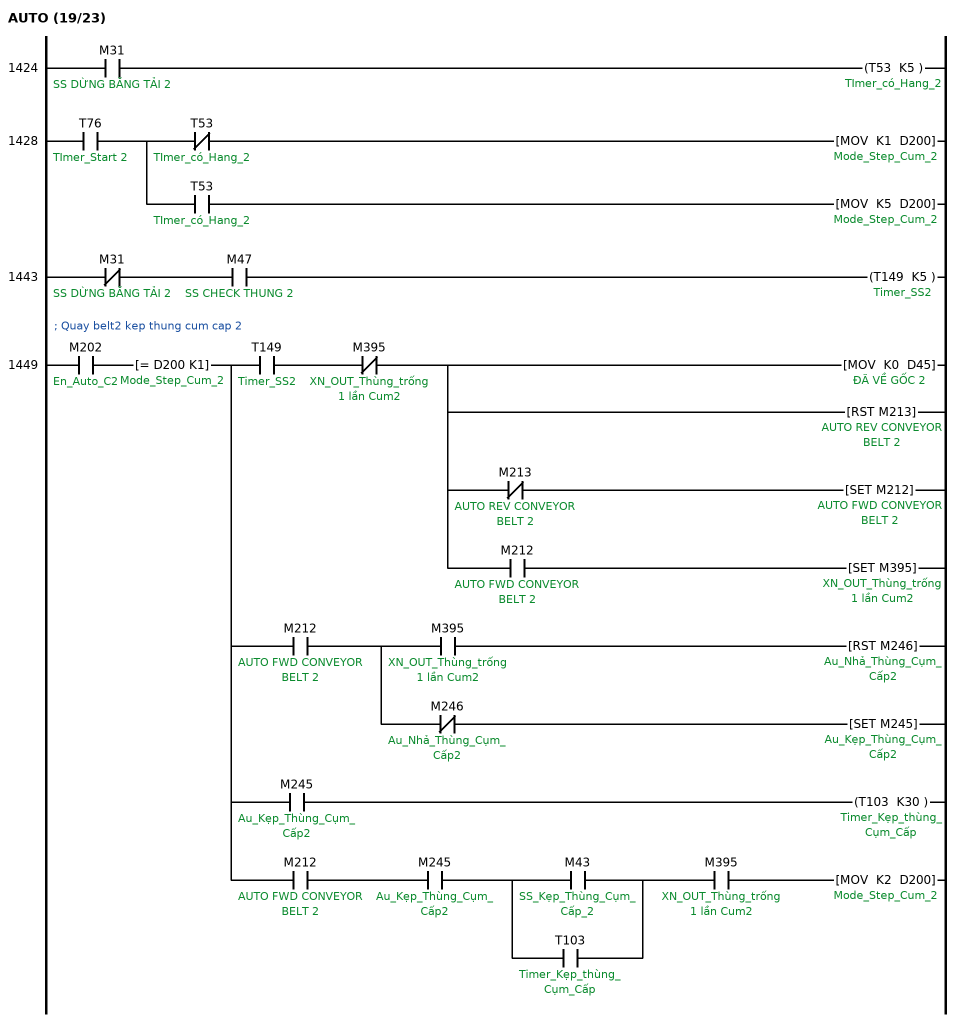
1424  LD      M31  ; SS DỪNG BĂNG TẢI 2
      OUT     T53 K5  ; TImer_có_Hang_2
1428  LD      T76  ; TImer_Start 2
      MPS
      ANI     T53  ; TImer_có_Hang_2
      MOV     K1 D200
      MPP
      AND     T53  ; TImer_có_Hang_2
      MOV     K5 D200
1443  LDI     M31  ; SS DỪNG BĂNG TẢI 2
      AND     M47  ; SS CHECK THUNG 2
      OUT     T149 K5  ; Timer_SS2
; Quay belt2 kep thung cum cap 2
1449  LD      M202  ; En_Auto_C2
      AND=    D200 K1  ; Mode_Step_Cum_2
      MPS
      AND     T149  ; Timer_SS2
      ANI     M395  ; XN_OUT_Thùng_trống 1 lần Cum2
      MOV     K0 D45
      RST     M213  ; AUTO REV CONVEYOR BELT 2
      MPS
      ANI     M213  ; AUTO REV CONVEYOR BELT 2
      SET     M212  ; AUTO FWD CONVEYOR BELT 2
      MPP
      AND     M212  ; AUTO FWD CONVEYOR BELT 2
      SET     M395  ; XN_OUT_Thùng_trống 1 lần Cum2
      MRD
      AND     M212  ; AUTO FWD CONVEYOR BELT 2
      MPS
      AND     M395  ; XN_OUT_Thùng_trống 1 lần Cum2
      RST     M246  ; Au_Nhả_Thùng_Cụm_Cấp2
      MPP
      ANI     M246  ; Au_Nhả_Thùng_Cụm_Cấp2
      SET     M245  ; Au_Kẹp_Thùng_Cụm_Cấp2
      MRD
      AND     M245  ; Au_Kẹp_Thùng_Cụm_Cấp2
      OUT     T103 K30  ; Timer_Kẹp_thùng_Cụm_Cấp
      MPP
      AND     M212  ; AUTO FWD CONVEYOR BELT 2
      AND     M245  ; Au_Kẹp_Thùng_Cụm_Cấp2
      LD      M43  ; SS_Kẹp_Thùng_Cụm_Cấp_2
      OR      T103  ; Timer_Kẹp_thùng_Cụm_Cấp
      ANB
      AND     M395  ; XN_OUT_Thùng_trống 1 lần Cum2
      MOV     K2 D200
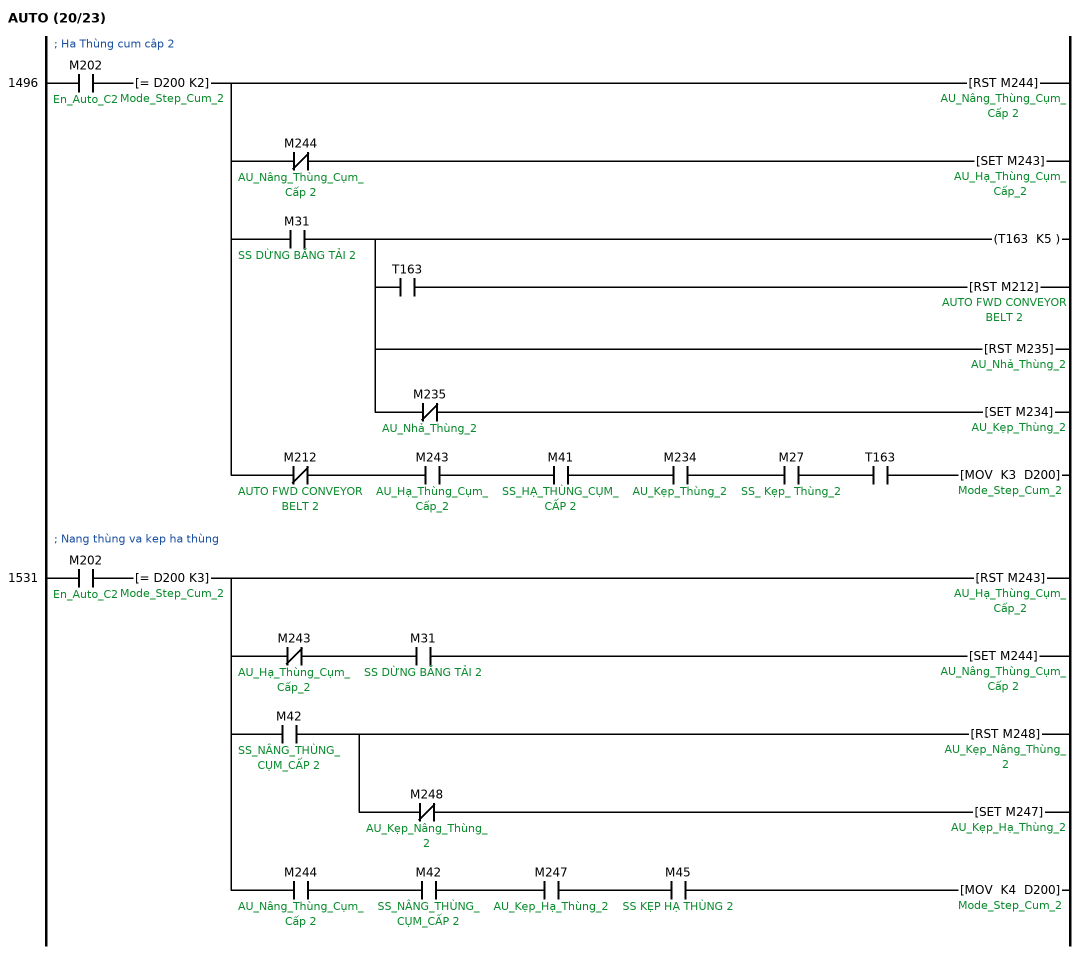
; Ha Thùng cum câp 2
1496  LD      M202  ; En_Auto_C2
      AND=    D200 K2  ; Mode_Step_Cum_2
      RST     M244  ; AU_Nâng_Thùng_Cụm_Cấp 2
      MPS
      ANI     M244  ; AU_Nâng_Thùng_Cụm_Cấp 2
      SET     M243  ; AU_Hạ_Thùng_Cụm_Cấp_2
      MRD
      AND     M31  ; SS DỪNG BĂNG TẢI 2
      OUT     T163 K5
      MPS
      AND     T163
      RST     M212  ; AUTO FWD CONVEYOR BELT 2
      MPP
      RST     M235  ; AU_Nhả_Thùng_2
      ANI     M235  ; AU_Nhả_Thùng_2
      SET     M234  ; AU_Kẹp_Thùng_2
      MPP
      ANI     M212  ; AUTO FWD CONVEYOR BELT 2
      AND     M243  ; AU_Hạ_Thùng_Cụm_Cấp_2
      AND     M41  ; SS_HẠ_THÙNG_CỤM_CẤP 2
      AND     M234  ; AU_Kẹp_Thùng_2
      AND     M27  ; SS_ Kẹp_ Thùng_2
      AND     T163
      MOV     K3 D200
; Nang thùng va kep ha thùng
1531  LD      M202  ; En_Auto_C2
      AND=    D200 K3  ; Mode_Step_Cum_2
      RST     M243  ; AU_Hạ_Thùng_Cụm_Cấp_2
      MPS
      ANI     M243  ; AU_Hạ_Thùng_Cụm_Cấp_2
      AND     M31  ; SS DỪNG BĂNG TẢI 2
      SET     M244  ; AU_Nâng_Thùng_Cụm_Cấp 2
      MRD
      AND     M42  ; SS_NÂNG_THÙNG_CỤM_CẤP 2
      RST     M248  ; AU_Kẹp_Nâng_Thùng_2
      ANI     M248  ; AU_Kẹp_Nâng_Thùng_2
      SET     M247  ; AU_Kẹp_Hạ_Thùng_2
      MPP
      AND     M244  ; AU_Nâng_Thùng_Cụm_Cấp 2
      AND     M42  ; SS_NÂNG_THÙNG_CỤM_CẤP 2
      AND     M247  ; AU_Kẹp_Hạ_Thùng_2
      AND     M45  ; SS KẸP HẠ THÙNG 2
      MOV     K4 D200
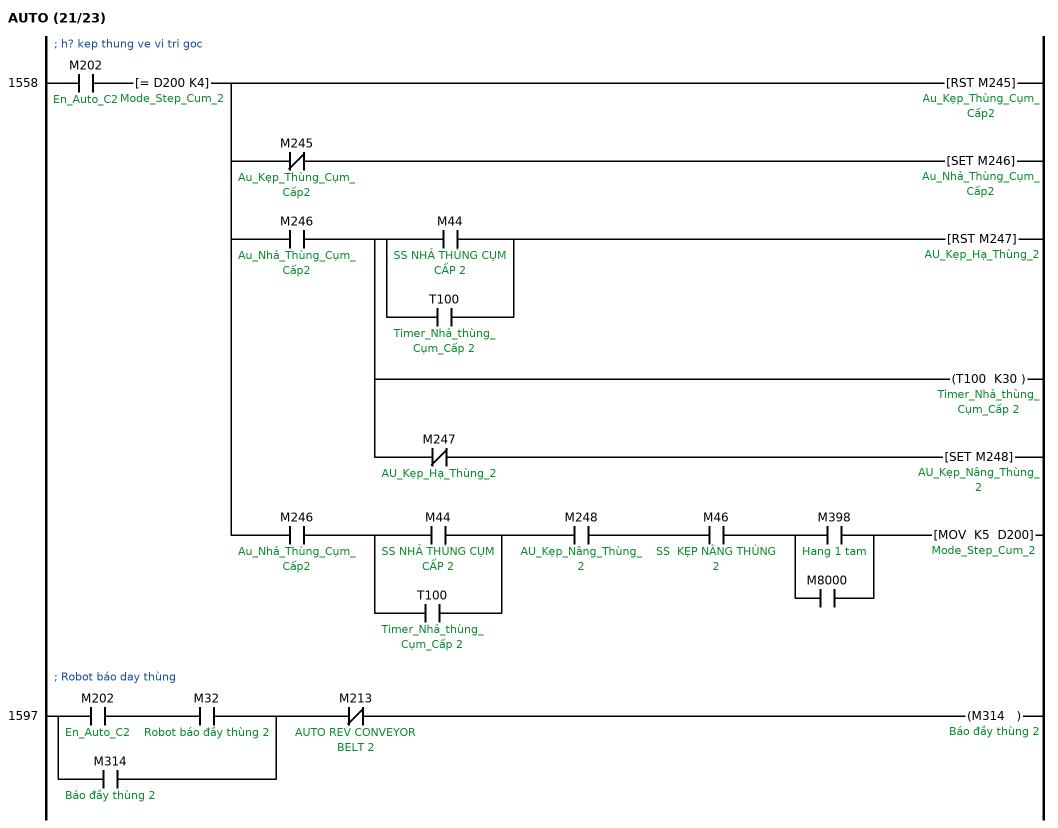
; h? kep thung ve vi tri goc
1558  LD      M202  ; En_Auto_C2
      AND=    D200 K4  ; Mode_Step_Cum_2
      RST     M245  ; Au_Kẹp_Thùng_Cụm_Cấp2
      MPS
      ANI     M245  ; Au_Kẹp_Thùng_Cụm_Cấp2
      SET     M246  ; Au_Nhả_Thùng_Cụm_Cấp2
      MRD
      AND     M246  ; Au_Nhả_Thùng_Cụm_Cấp2
      MPS
      LD      M44  ; SS NHẢ THÙNG CỤM CẤP 2
      OR      T100  ; Timer_Nhả_thùng_Cụm_Cấp 2
      ANB
      RST     M247  ; AU_Kẹp_Hạ_Thùng_2
      MPP
      OUT     T100 K30  ; Timer_Nhả_thùng_Cụm_Cấp 2
      ANI     M247  ; AU_Kẹp_Hạ_Thùng_2
      SET     M248  ; AU_Kẹp_Nâng_Thùng_2
      MPP
      AND     M246  ; Au_Nhả_Thùng_Cụm_Cấp2
      LD      M44  ; SS NHẢ THÙNG CỤM CẤP 2
      OR      T100  ; Timer_Nhả_thùng_Cụm_Cấp 2
      ANB
      AND     M248  ; AU_Kẹp_Nâng_Thùng_2
      AND     M46  ; SS  KẸP NÂNG THÙNG 2
      LD      M398  ; Hang 1 tam
      OR      M8000
      ANB
      MOV     K5 D200
; Robot báo day thùng
1597  LD      M202  ; En_Auto_C2
      AND     M32  ; Robot báo đầy thùng 2
      OR      M314  ; Báo đầy thùng 2
      ANI     M213  ; AUTO REV CONVEYOR BELT 2
      OUT     M314  ; Báo đầy thùng 2
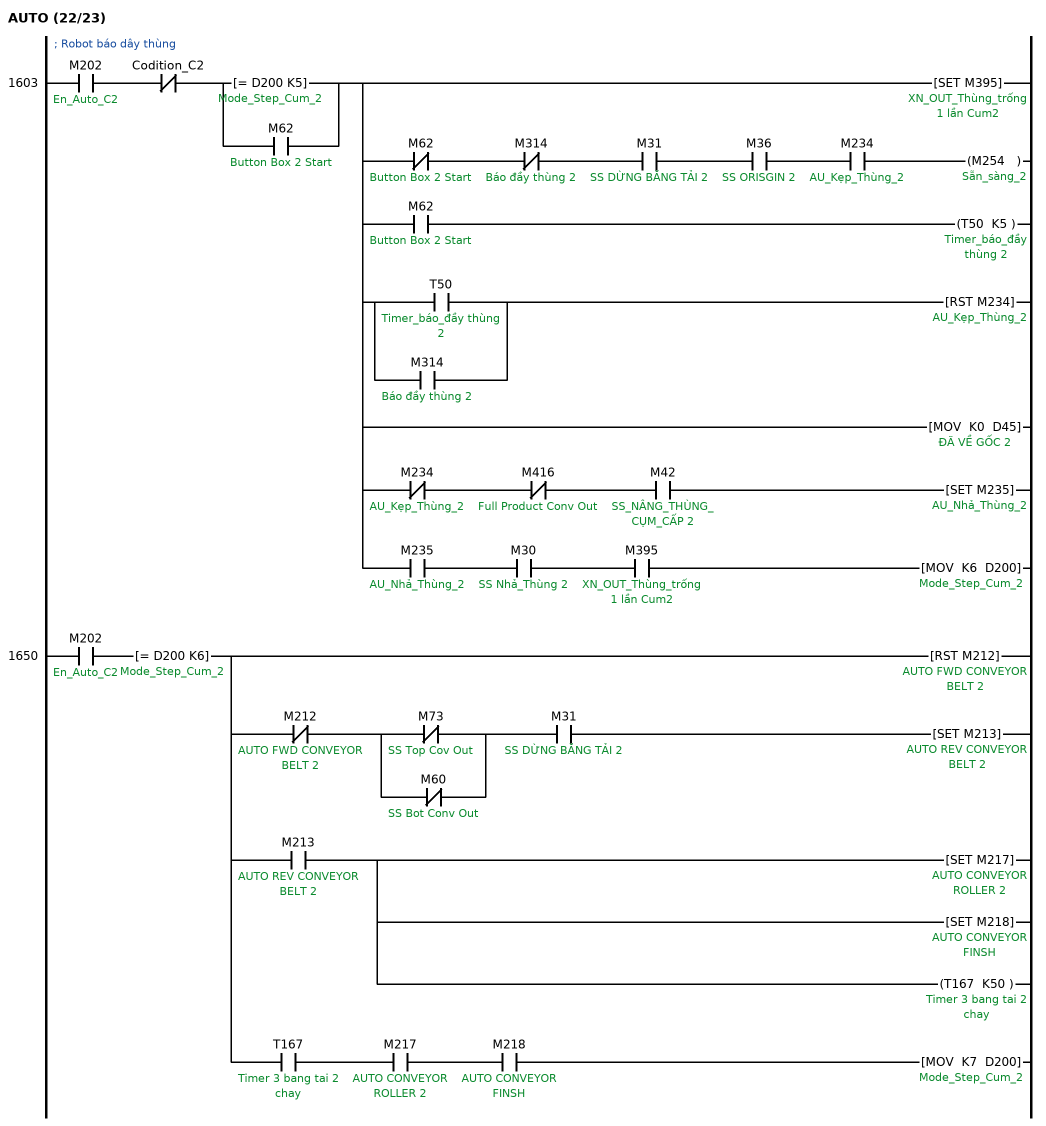
; Robot báo dây thùng
1603  LD      M202  ; En_Auto_C2
      ANI     Codition_C2
      LD=     D200 K5  ; Mode_Step_Cum_2
      OR      M62  ; Button Box 2 Start
      ANB
      SET     M395  ; XN_OUT_Thùng_trống 1 lần Cum2
      MPS
      ANI     M62  ; Button Box 2 Start
      ANI     M314  ; Báo đầy thùng 2
      AND     M31  ; SS DỪNG BĂNG TẢI 2
      AND     M36  ; SS ORISGIN 2
      AND     M234  ; AU_Kẹp_Thùng_2
      OUT     M254  ; Sẵn_sàng_2
      MRD
      AND     M62  ; Button Box 2 Start
      OUT     T50 K5  ; Timer_báo_đầy thùng 2
      MRD
      LD      T50  ; Timer_báo_đầy thùng 2
      OR      M314  ; Báo đầy thùng 2
      ANB
      RST     M234  ; AU_Kẹp_Thùng_2
      MPP
      MOV     K0 D45
      MPS
      ANI     M234  ; AU_Kẹp_Thùng_2
      ANI     M416  ; Full Product Conv Out
      AND     M42  ; SS_NÂNG_THÙNG_CỤM_CẤP 2
      SET     M235  ; AU_Nhả_Thùng_2
      MPP
      AND     M235  ; AU_Nhả_Thùng_2
      AND     M30  ; SS Nhả_Thùng 2
      AND     M395  ; XN_OUT_Thùng_trống 1 lần Cum2
      MOV     K6 D200
1650  LD      M202  ; En_Auto_C2
      AND=    D200 K6  ; Mode_Step_Cum_2
      RST     M212  ; AUTO FWD CONVEYOR BELT 2
      MPS
      ANI     M212  ; AUTO FWD CONVEYOR BELT 2
      LDI     M73  ; SS Top Cov Out
      ORI     M60  ; SS Bot Conv Out
      ANB
      AND     M31  ; SS DỪNG BĂNG TẢI 2
      SET     M213  ; AUTO REV CONVEYOR BELT 2
      MRD
      AND     M213  ; AUTO REV CONVEYOR BELT 2
      SET     M217  ; AUTO CONVEYOR ROLLER 2
      SET     M218  ; AUTO CONVEYOR FINSH
      OUT     T167 K50  ; Timer 3 bang tai 2 chay
      MPP
      AND     T167  ; Timer 3 bang tai 2 chay
      AND     M217  ; AUTO CONVEYOR ROLLER 2
      AND     M218  ; AUTO CONVEYOR FINSH
      MOV     K7 D200
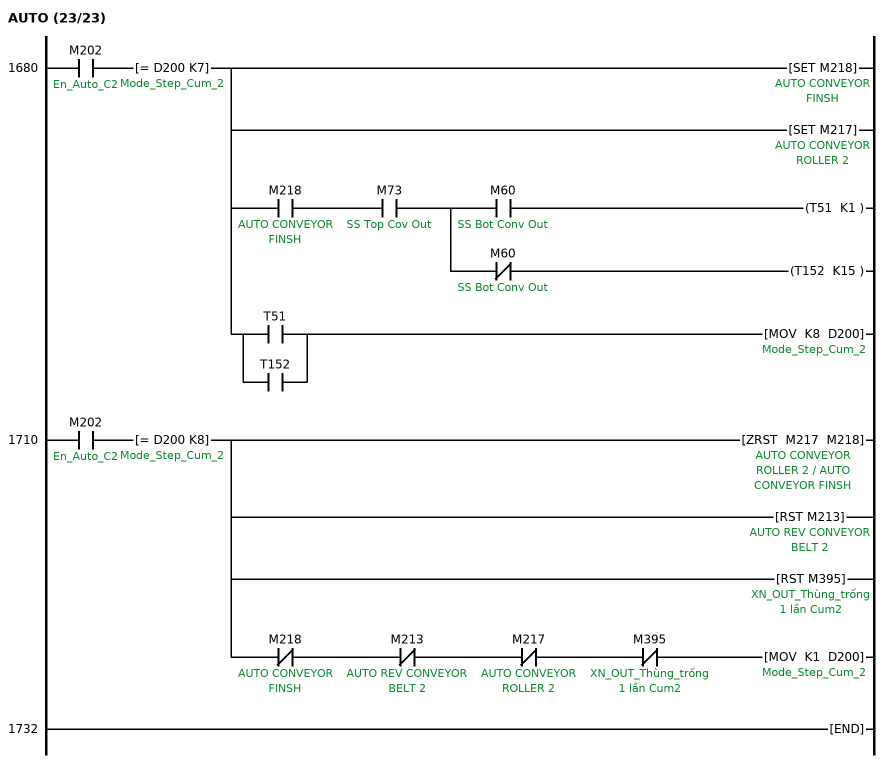
1680  LD      M202  ; En_Auto_C2
      AND=    D200 K7  ; Mode_Step_Cum_2
      SET     M218  ; AUTO CONVEYOR FINSH
      SET     M217  ; AUTO CONVEYOR ROLLER 2
      MPS
      AND     M218  ; AUTO CONVEYOR FINSH
      AND     M73  ; SS Top Cov Out
      MPS
      AND     M60  ; SS Bot Conv Out
      OUT     T51 K1
      MPP
      ANI     M60  ; SS Bot Conv Out
      OUT     T152 K15
      MPP
      LD      T51
      OR      T152
      ANB
      MOV     K8 D200
1710  LD      M202  ; En_Auto_C2
      AND=    D200 K8  ; Mode_Step_Cum_2
      ZRST    M217 M218
      RST     M213  ; AUTO REV CONVEYOR BELT 2
      RST     M395  ; XN_OUT_Thùng_trống 1 lần Cum2
      ANI     M218  ; AUTO CONVEYOR FINSH
      ANI     M213  ; AUTO REV CONVEYOR BELT 2
      ANI     M217  ; AUTO CONVEYOR ROLLER 2
      ANI     M395  ; XN_OUT_Thùng_trống 1 lần Cum2
      MOV     K1 D200
1732  END
END_PROGRAM

PROGRAM Auxil
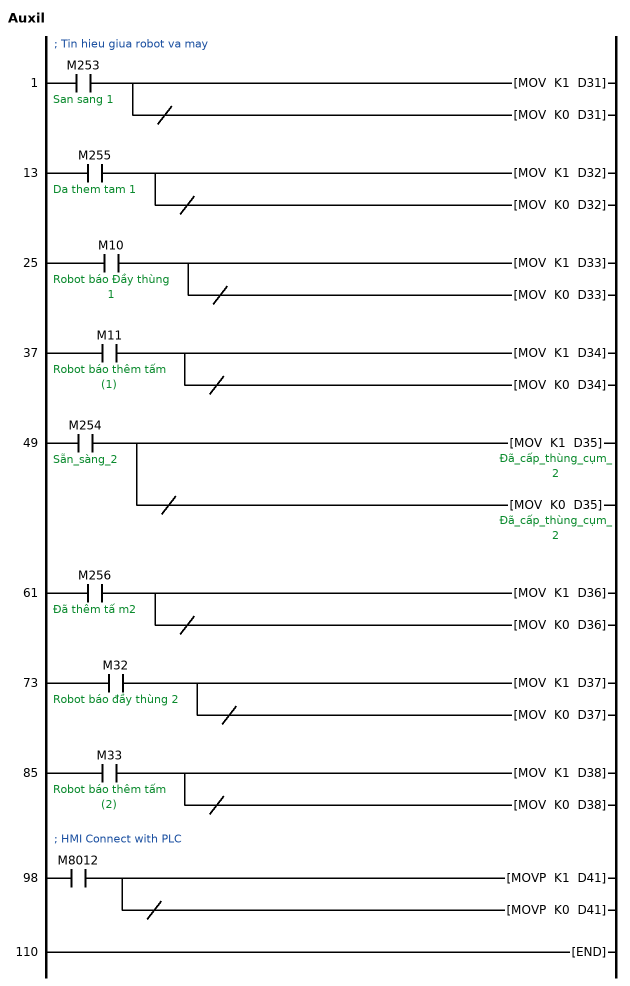
; Tin hieu giua robot va may
1     LD      M253  ; San sang 1
      MOV     K1 D31
      INV
      MOV     K0 D31
13    LD      M255  ; Da them tam 1
      MOV     K1 D32
      INV
      MOV     K0 D32
25    LD      M10  ; Robot báo Đầy thùng 1
      MOV     K1 D33
      INV
      MOV     K0 D33
37    LD      M11  ; Robot báo thêm tấm (1)
      MOV     K1 D34
      INV
      MOV     K0 D34
49    LD      M254  ; Sẵn_sàng_2
      MOV     K1 D35  ; Đã_cấp_thùng_cụm_2
      INV
      MOV     K0 D35
61    LD      M256  ; Đã thêm tấ m2
      MOV     K1 D36
      INV
      MOV     K0 D36
73    LD      M32  ; Robot báo đầy thùng 2
      MOV     K1 D37
      INV
      MOV     K0 D37
85    LD      M33  ; Robot báo thêm tấm (2)
      MOV     K1 D38
      INV
      MOV     K0 D38
; HMI Connect with PLC
98    LD      M8012
      MOVP    K1 D41
      INV
      MOVP    K0 D41
110   END
END_PROGRAM

PROGRAM INPUT
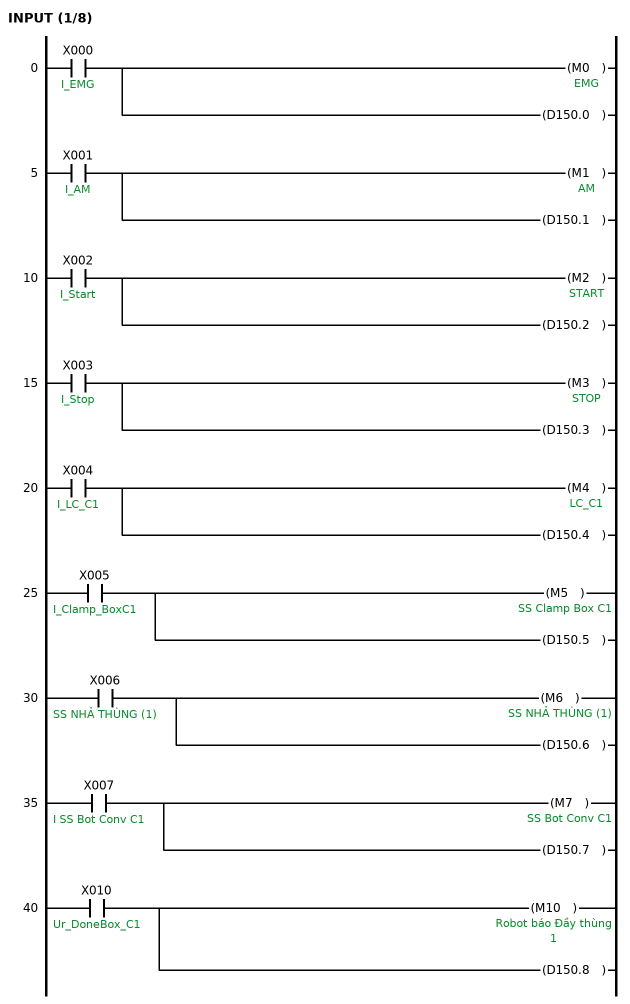
0     LD      X000  ; I_EMG
      OUT     M0  ; EMG
      OUT     D150.0
5     LD      X001  ; I_AM
      OUT     M1  ; AM
      OUT     D150.1
10    LD      X002  ; I_Start
      OUT     M2  ; START
      OUT     D150.2
15    LD      X003  ; I_Stop
      OUT     M3  ; STOP
      OUT     D150.3
20    LD      X004  ; I_LC_C1
      OUT     M4  ; LC_C1
      OUT     D150.4
25    LD      X005  ; I_Clamp_BoxC1
      OUT     M5  ; SS Clamp Box C1
      OUT     D150.5
30    LD      X006  ; SS NHẢ THÙNG (1)
      OUT     M6  ; SS NHẢ THÙNG (1)
      OUT     D150.6
35    LD      X007  ; I SS Bot Conv C1
      OUT     M7  ; SS Bot Conv C1
      OUT     D150.7
40    LD      X010  ; Ur_DoneBox_C1
      OUT     M10  ; Robot báo Đầy thùng 1
      OUT     D150.8
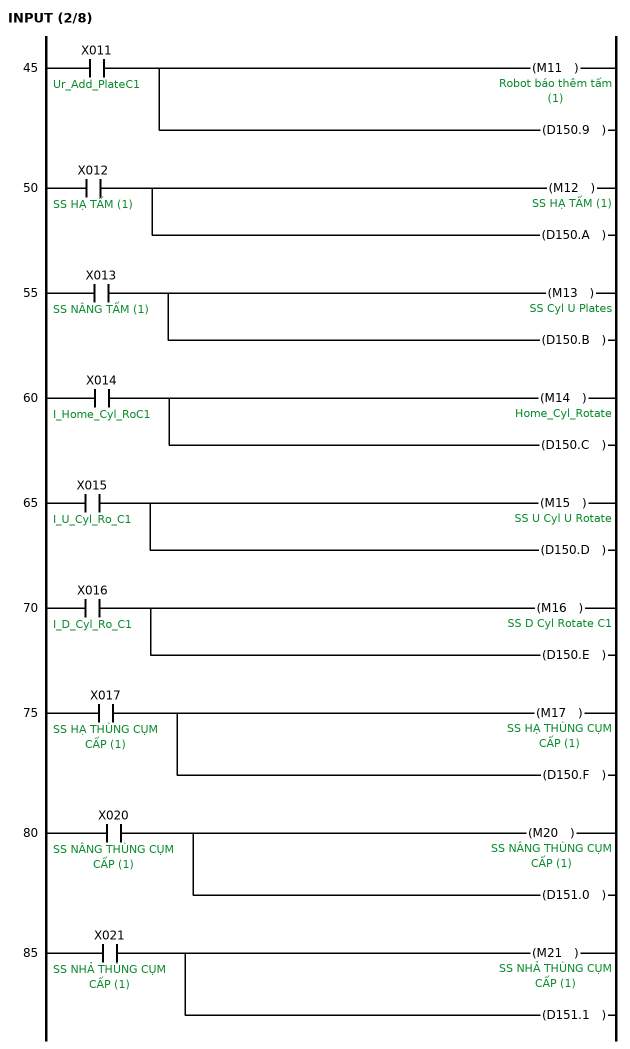
45    LD      X011  ; Ur_Add_PlateC1
      OUT     M11  ; Robot báo thêm tấm (1)
      OUT     D150.9
50    LD      X012  ; SS HẠ TẤM (1)
      OUT     M12  ; SS HẠ TẤM (1)
      OUT     D150.A
55    LD      X013  ; SS NÂNG TẤM (1)
      OUT     M13  ; SS Cyl U Plates
      OUT     D150.B
60    LD      X014  ; I_Home_Cyl_RoC1
      OUT     M14  ; Home_Cyl_Rotate
      OUT     D150.C
65    LD      X015  ; I_U_Cyl_Ro_C1
      OUT     M15  ; SS U Cyl U Rotate
      OUT     D150.D
70    LD      X016  ; I_D_Cyl_Ro_C1
      OUT     M16  ; SS D Cyl Rotate C1
      OUT     D150.E
75    LD      X017  ; SS HẠ THÙNG CỤM CẤP (1)
      OUT     M17  ; SS HẠ THÙNG CỤM CẤP (1)
      OUT     D150.F
80    LD      X020  ; SS NÂNG THÙNG CỤM CẤP (1)
      OUT     M20  ; SS NÂNG THÙNG CỤM CẤP (1)
      OUT     D151.0
85    LD      X021  ; SS NHẢ THÙNG CỤM CẤP (1)
      OUT     M21  ; SS NHẢ THÙNG CỤM CẤP (1)
      OUT     D151.1
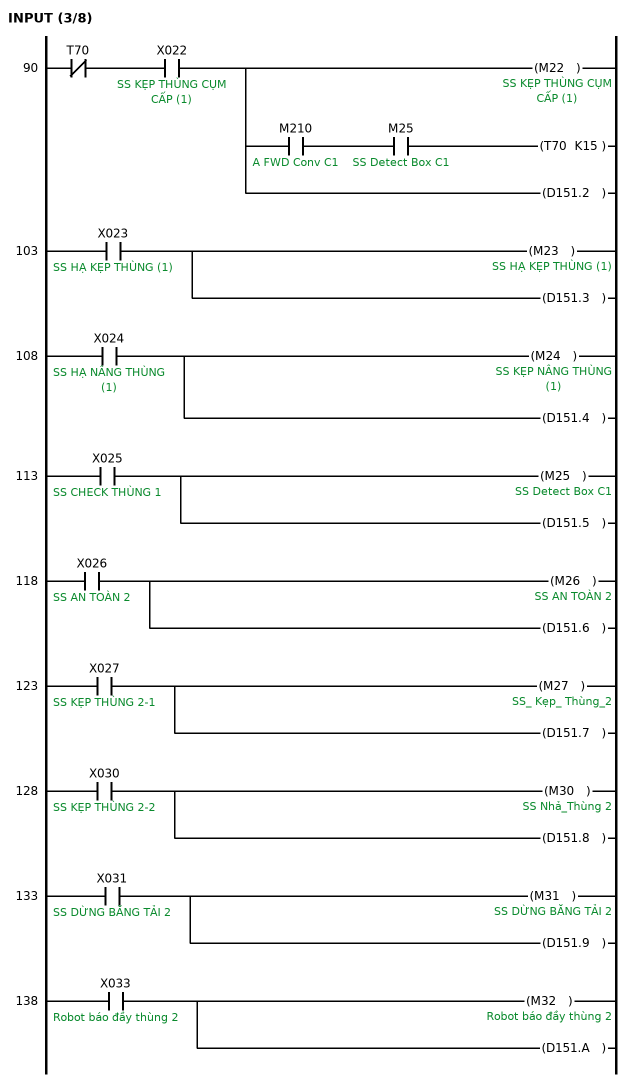
90    LDI     T70
      AND     X022  ; SS KẸP THÙNG CỤM CẤP (1)
      OUT     M22  ; SS KẸP THÙNG CỤM CẤP (1)
      MPS
      AND     M210  ; A FWD Conv C1
      AND     M25  ; SS Detect Box C1
      OUT     T70 K15
      MPP
      OUT     D151.2
103   LD      X023  ; SS HẠ KẸP THÙNG (1)
      OUT     M23  ; SS HẠ KẸP THÙNG (1)
      OUT     D151.3
108   LD      X024  ; SS HẠ NÂNG THÙNG (1)
      OUT     M24  ; SS KẸP NÂNG THÙNG (1)
      OUT     D151.4
113   LD      X025  ; SS CHECK THÙNG 1
      OUT     M25  ; SS Detect Box C1
      OUT     D151.5
118   LD      X026  ; SS AN TOÀN 2
      OUT     M26  ; SS AN TOÀN 2
      OUT     D151.6
123   LD      X027  ; SS KẸP THÙNG 2-1
      OUT     M27  ; SS_ Kẹp_ Thùng_2
      OUT     D151.7
128   LD      X030  ; SS KẸP THÙNG 2-2
      OUT     M30  ; SS Nhả_Thùng 2
      OUT     D151.8
133   LD      X031  ; SS DỪNG BĂNG TẢI 2
      OUT     M31  ; SS DỪNG BĂNG TẢI 2
      OUT     D151.9
138   LD      X033  ; Robot báo đầy thùng 2
      OUT     M32  ; Robot báo đầy thùng 2
      OUT     D151.A
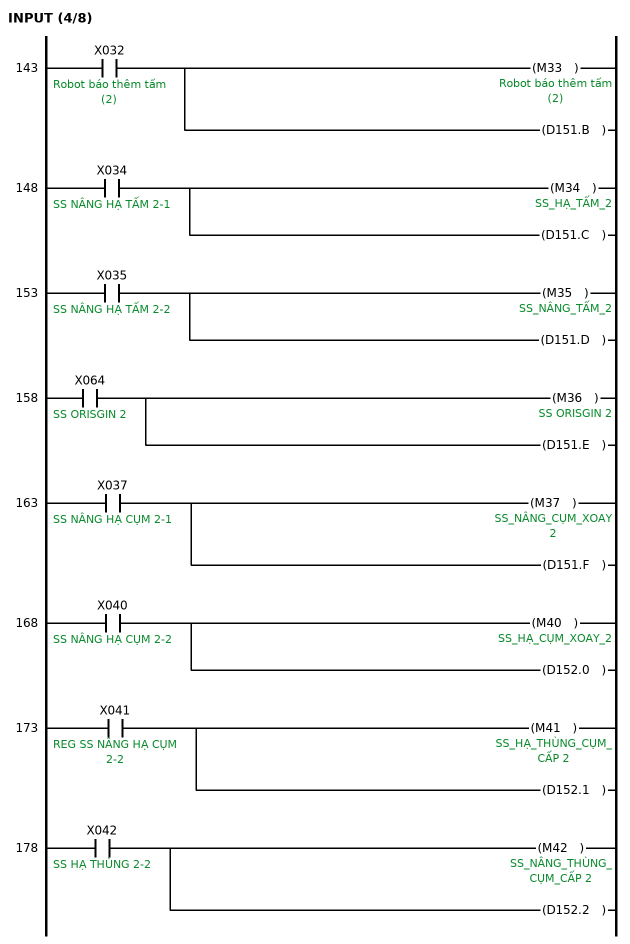
143   LD      X032  ; Robot báo thêm tấm (2)
      OUT     M33  ; Robot báo thêm tấm (2)
      OUT     D151.B
148   LD      X034  ; SS NÂNG HẠ TẤM 2-1
      OUT     M34  ; SS_HẠ_TẤM_2
      OUT     D151.C
153   LD      X035  ; SS NÂNG HẠ TẤM 2-2
      OUT     M35  ; SS_NÂNG_TẤM_2
      OUT     D151.D
158   LD      X064  ; SS ORISGIN 2
      OUT     M36  ; SS ORISGIN 2
      OUT     D151.E
163   LD      X037  ; SS NÂNG HẠ CỤM 2-1
      OUT     M37  ; SS_NÂNG_CỤM_XOAY 2
      OUT     D151.F
168   LD      X040  ; SS NÂNG HẠ CỤM 2-2
      OUT     M40  ; SS_HẠ_CỤM_XOAY_2
      OUT     D152.0
173   LD      X041  ; REG SS NÂNG HẠ CỤM 2-2
      OUT     M41  ; SS_HẠ_THÙNG_CỤM_CẤP 2
      OUT     D152.1
178   LD      X042  ; SS HẠ THÙNG 2-2
      OUT     M42  ; SS_NÂNG_THÙNG_CỤM_CẤP 2
      OUT     D152.2
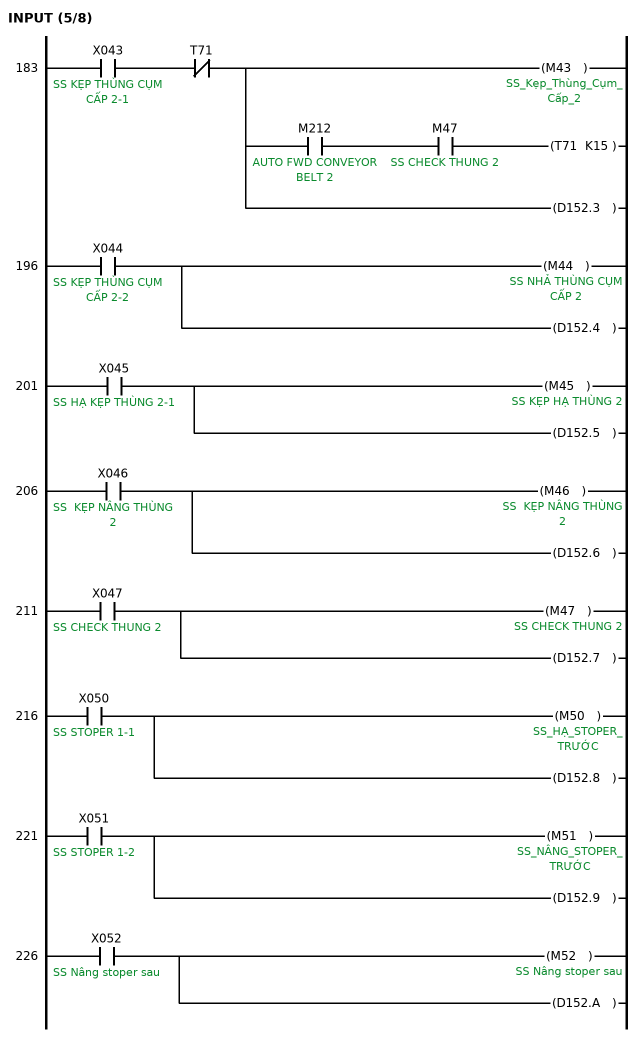
183   LD      X043  ; SS KẸP THÙNG CỤM CẤP 2-1
      ANI     T71
      OUT     M43  ; SS_Kẹp_Thùng_Cụm_Cấp_2
      MPS
      AND     M212  ; AUTO FWD CONVEYOR BELT 2
      AND     M47  ; SS CHECK THUNG 2
      OUT     T71 K15
      MPP
      OUT     D152.3
196   LD      X044  ; SS KẸP THÙNG CỤM CẤP 2-2
      OUT     M44  ; SS NHẢ THÙNG CỤM CẤP 2
      OUT     D152.4
201   LD      X045  ; SS HẠ KẸP THÙNG 2-1
      OUT     M45  ; SS KẸP HẠ THÙNG 2
      OUT     D152.5
206   LD      X046  ; SS  KẸP NÂNG THÙNG 2
      OUT     M46  ; SS  KẸP NÂNG THÙNG 2
      OUT     D152.6
211   LD      X047  ; SS CHECK THUNG 2
      OUT     M47  ; SS CHECK THUNG 2
      OUT     D152.7
216   LD      X050  ; SS STOPER 1-1
      OUT     M50  ; SS_HẠ_STOPER_TRƯỚC
      OUT     D152.8
221   LD      X051  ; SS STOPER 1-2
      OUT     M51  ; SS_NÂNG_STOPER_TRƯỚC
      OUT     D152.9
226   LD      X052  ; SS Nâng stoper sau
      OUT     M52  ; SS Nâng stoper sau
      OUT     D152.A
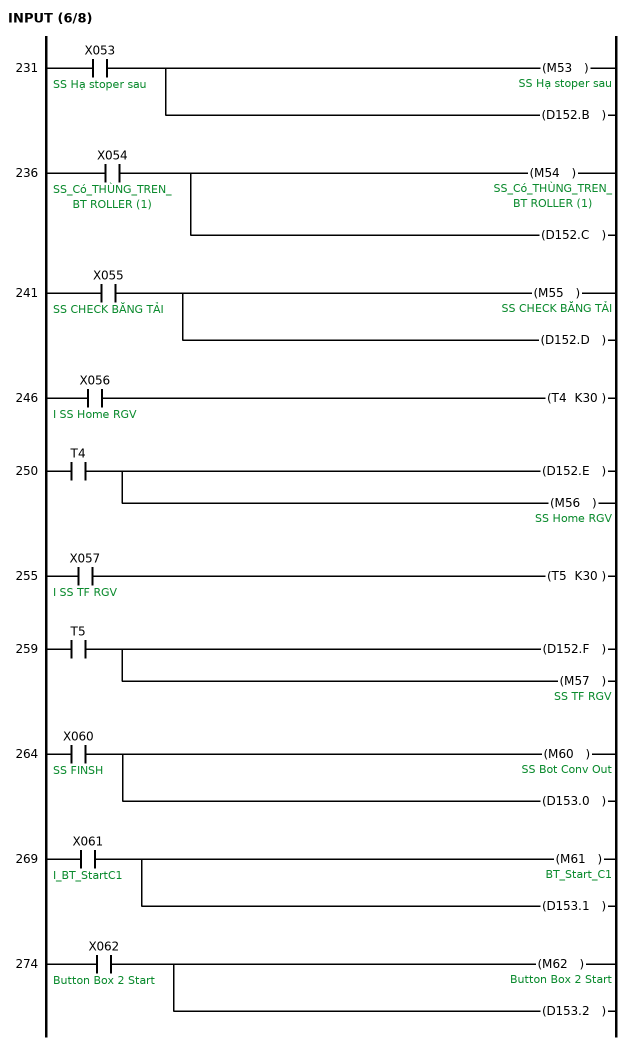
231   LD      X053  ; SS Hạ stoper sau
      OUT     M53  ; SS Hạ stoper sau
      OUT     D152.B
236   LD      X054  ; SS_Có_THÙNG_TREN_BT ROLLER (1)
      OUT     M54  ; SS_Có_THÙNG_TREN_BT ROLLER (1)
      OUT     D152.C
241   LD      X055  ; SS CHECK BĂNG TẢI
      OUT     M55  ; SS CHECK BĂNG TẢI
      OUT     D152.D
246   LD      X056  ; I SS Home RGV
      OUT     T4 K30
250   LD      T4
      OUT     D152.E
      OUT     M56  ; SS Home RGV
255   LD      X057  ; I SS TF RGV
      OUT     T5 K30
259   LD      T5
      OUT     D152.F
      OUT     M57  ; SS TF RGV
264   LD      X060  ; SS FINSH
      OUT     M60  ; SS Bot Conv Out
      OUT     D153.0
269   LD      X061  ; I_BT_StartC1
      OUT     M61  ; BT_Start_C1
      OUT     D153.1
274   LD      X062  ; Button Box 2 Start
      OUT     M62  ; Button Box 2 Start
      OUT     D153.2
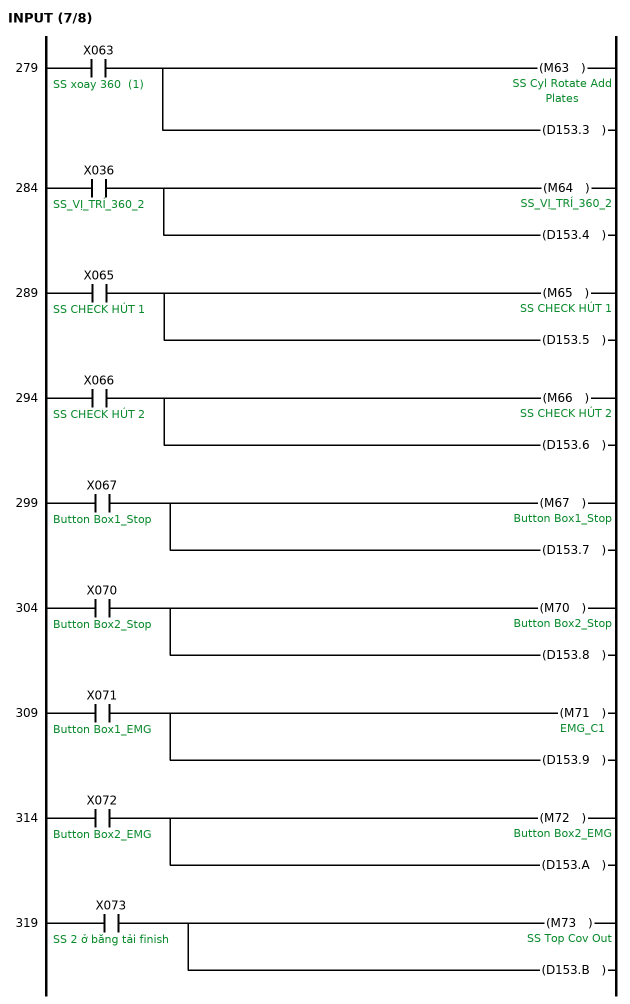
279   LD      X063  ; SS xoay 360  (1)
      OUT     M63  ; SS Cyl Rotate Add Plates
      OUT     D153.3
284   LD      X036  ; SS_VỊ_TRÍ_360_2
      OUT     M64  ; SS_VỊ_TRÍ_360_2
      OUT     D153.4
289   LD      X065  ; SS CHECK HÚT 1
      OUT     M65  ; SS CHECK HÚT 1
      OUT     D153.5
294   LD      X066  ; SS CHECK HÚT 2
      OUT     M66  ; SS CHECK HÚT 2
      OUT     D153.6
299   LD      X067  ; Button Box1_Stop
      OUT     M67  ; Button Box1_Stop
      OUT     D153.7
304   LD      X070  ; Button Box2_Stop
      OUT     M70  ; Button Box2_Stop
      OUT     D153.8
309   LD      X071  ; Button Box1_EMG
      OUT     M71  ; EMG_C1
      OUT     D153.9
314   LD      X072  ; Button Box2_EMG
      OUT     M72  ; Button Box2_EMG
      OUT     D153.A
319   LD      X073  ; SS 2 ở băng tải finish
      OUT     M73  ; SS Top Cov Out
      OUT     D153.B
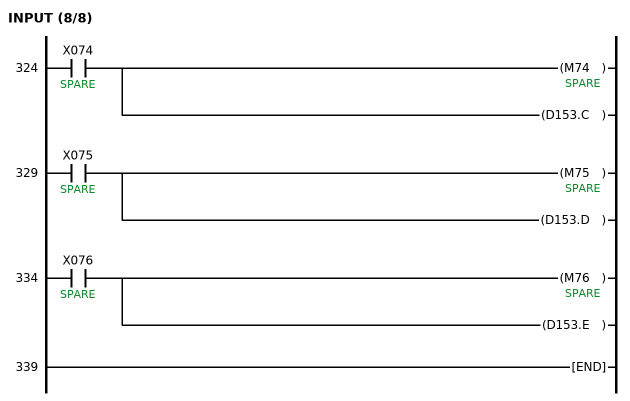
324   LD      X074  ; SPARE
      OUT     M74  ; SPARE
      OUT     D153.C
329   LD      X075  ; SPARE
      OUT     M75  ; SPARE
      OUT     D153.D
334   LD      X076  ; SPARE
      OUT     M76  ; SPARE
      OUT     D153.E
339   END
END_PROGRAM

PROGRAM OUTPUT
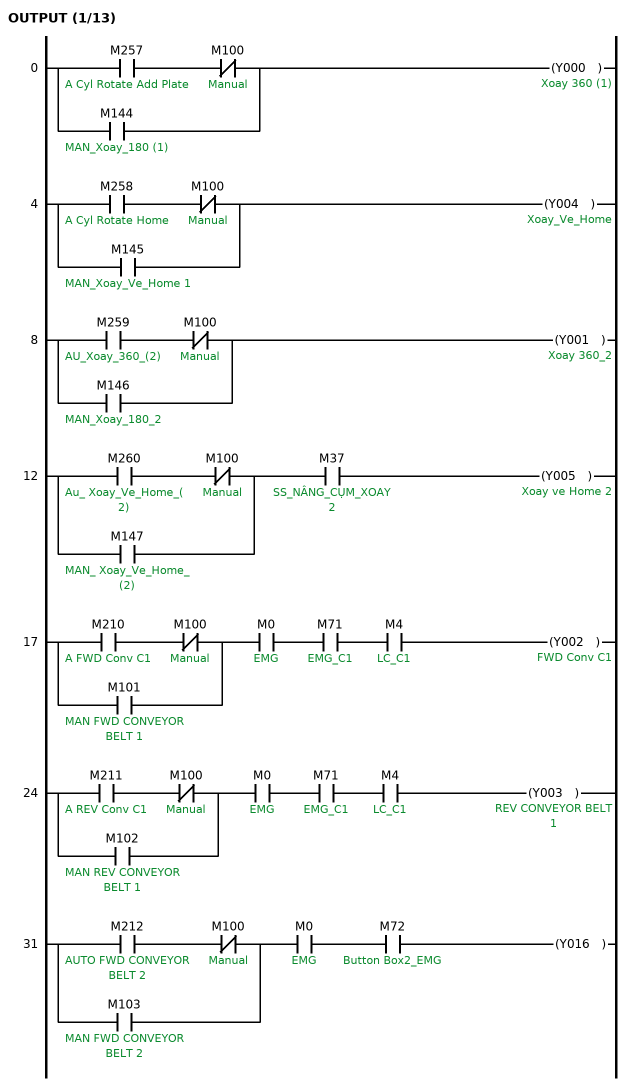
0     LD      M257  ; A Cyl Rotate Add Plate
      ANI     M100  ; Manual
      OR      M144  ; MAN_Xoay_180 (1)
      OUT     Y000  ; Xoay 360 (1)
4     LD      M258  ; A Cyl Rotate Home
      ANI     M100  ; Manual
      OR      M145  ; MAN_Xoay_Ve_Home 1
      OUT     Y004  ; Xoay_Ve_Home
8     LD      M259  ; AU_Xoay_360_(2)
      ANI     M100  ; Manual
      OR      M146  ; MAN_Xoay_180_2
      OUT     Y001  ; Xoay 360_2
12    LD      M260  ; Au_ Xoay_Ve_Home_(2)
      ANI     M100  ; Manual
      OR      M147  ; MAN_ Xoay_Ve_Home_(2)
      AND     M37  ; SS_NÂNG_CỤM_XOAY 2
      OUT     Y005  ; Xoay ve Home 2
17    LD      M210  ; A FWD Conv C1
      ANI     M100  ; Manual
      OR      M101  ; MAN FWD CONVEYOR BELT 1
      AND     M0  ; EMG
      AND     M71  ; EMG_C1
      AND     M4  ; LC_C1
      OUT     Y002  ; FWD Conv C1
24    LD      M211  ; A REV Conv C1
      ANI     M100  ; Manual
      OR      M102  ; MAN REV CONVEYOR BELT 1
      AND     M0  ; EMG
      AND     M71  ; EMG_C1
      AND     M4  ; LC_C1
      OUT     Y003  ; REV CONVEYOR BELT 1
31    LD      M212  ; AUTO FWD CONVEYOR BELT 2
      ANI     M100  ; Manual
      OR      M103  ; MAN FWD CONVEYOR BELT 2
      AND     M0  ; EMG
      AND     M72  ; Button Box2_EMG
      OUT     Y016
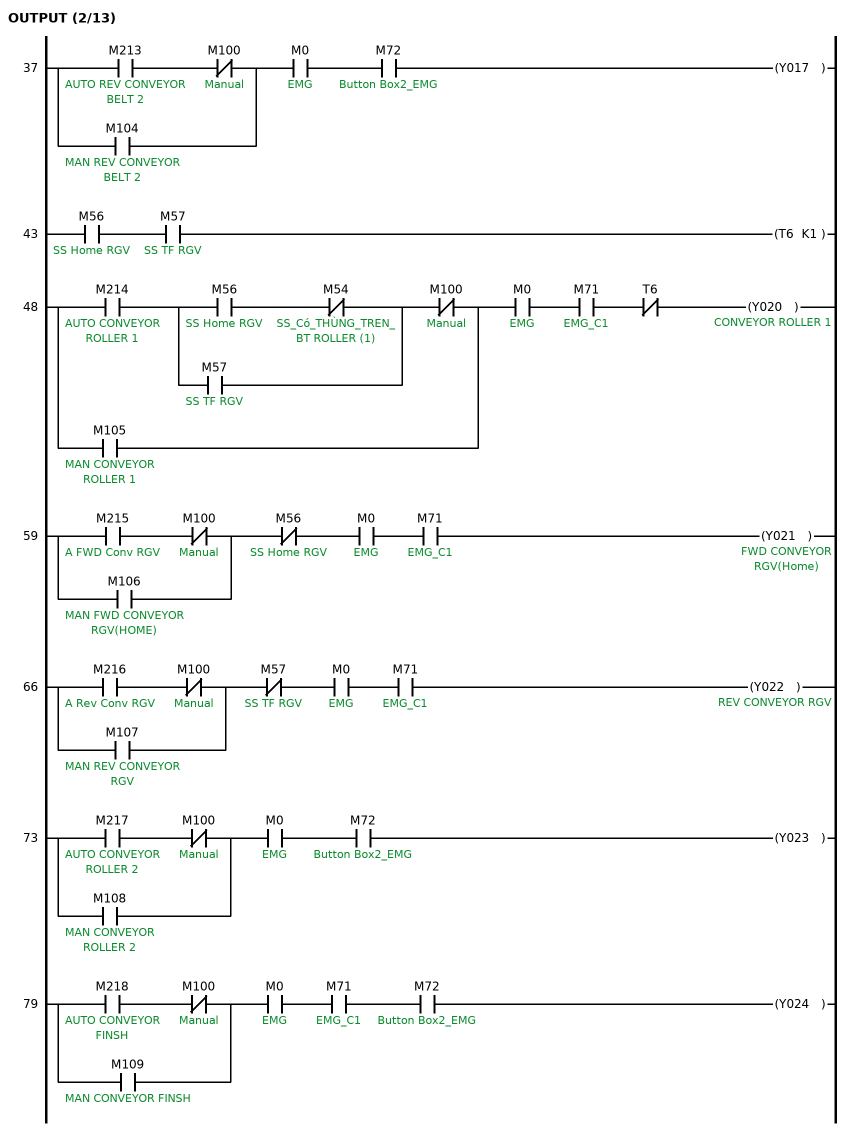
37    LD      M213  ; AUTO REV CONVEYOR BELT 2
      ANI     M100  ; Manual
      OR      M104  ; MAN REV CONVEYOR BELT 2
      AND     M0  ; EMG
      AND     M72  ; Button Box2_EMG
      OUT     Y017
43    LD      M56  ; SS Home RGV
      AND     M57  ; SS TF RGV
      OUT     T6 K1
48    LD      M214  ; AUTO CONVEYOR ROLLER 1
      LD      M56  ; SS Home RGV
      ANI     M54  ; SS_Có_THÙNG_TREN_BT ROLLER (1)
      OR      M57  ; SS TF RGV
      ANB
      ANI     M100  ; Manual
      OR      M105  ; MAN CONVEYOR ROLLER 1
      AND     M0  ; EMG
      AND     M71  ; EMG_C1
      ANI     T6
      OUT     Y020  ; CONVEYOR ROLLER 1
59    LD      M215  ; A FWD Conv RGV
      ANI     M100  ; Manual
      OR      M106  ; MAN FWD CONVEYOR RGV(HOME)
      ANI     M56  ; SS Home RGV
      AND     M0  ; EMG
      AND     M71  ; EMG_C1
      OUT     Y021  ; FWD CONVEYOR RGV(Home)
66    LD      M216  ; A Rev Conv RGV
      ANI     M100  ; Manual
      OR      M107  ; MAN REV CONVEYOR RGV
      ANI     M57  ; SS TF RGV
      AND     M0  ; EMG
      AND     M71  ; EMG_C1
      OUT     Y022  ; REV CONVEYOR RGV
73    LD      M217  ; AUTO CONVEYOR ROLLER 2
      ANI     M100  ; Manual
      OR      M108  ; MAN CONVEYOR ROLLER 2
      AND     M0  ; EMG
      AND     M72  ; Button Box2_EMG
      OUT     Y023
79    LD      M218  ; AUTO CONVEYOR FINSH
      ANI     M100  ; Manual
      OR      M109  ; MAN CONVEYOR FINSH
      AND     M0  ; EMG
      AND     M71  ; EMG_C1
      AND     M72  ; Button Box2_EMG
      OUT     Y024
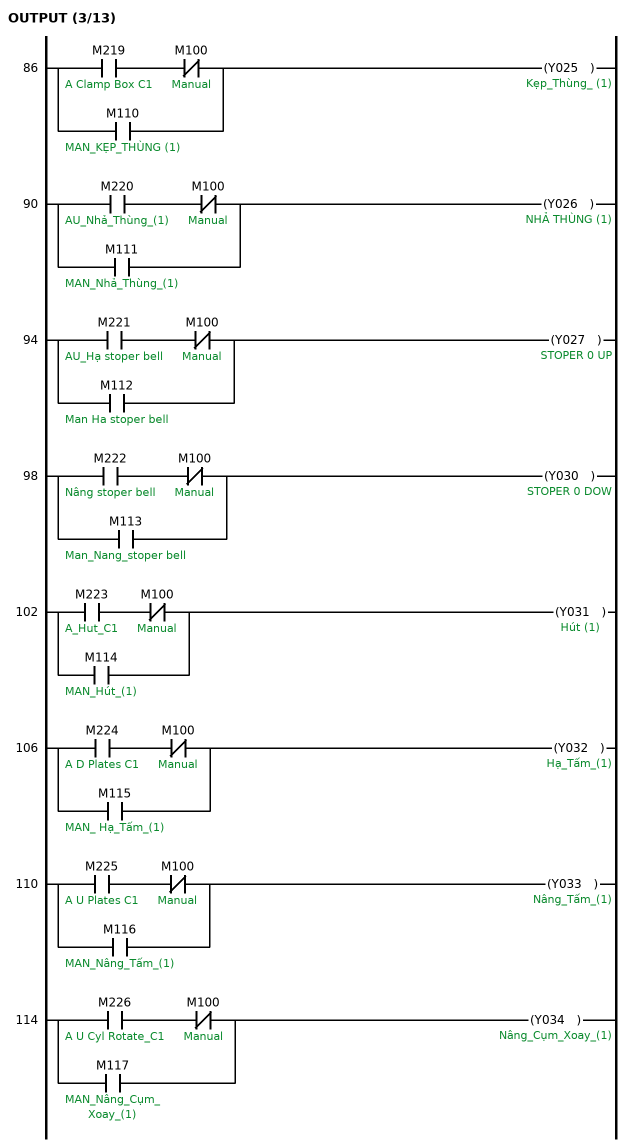
86    LD      M219  ; A Clamp Box C1
      ANI     M100  ; Manual
      OR      M110  ; MAN_KẸP_THÙNG (1)
      OUT     Y025  ; Kẹp_Thùng_ (1)
90    LD      M220  ; AU_Nhả_Thùng_(1)
      ANI     M100  ; Manual
      OR      M111  ; MAN_Nhả_Thùng_(1)
      OUT     Y026  ; NHẢ THÙNG (1)
94    LD      M221  ; AU_Hạ stoper bell
      ANI     M100  ; Manual
      OR      M112  ; Man Ha stoper bell
      OUT     Y027  ; STOPER 0 UP
98    LD      M222  ; Nâng stoper bell
      ANI     M100  ; Manual
      OR      M113  ; Man_Nang_stoper bell
      OUT     Y030  ; STOPER 0 DOW
102   LD      M223  ; A_Hut_C1
      ANI     M100  ; Manual
      OR      M114  ; MAN_Hút_(1)
      OUT     Y031  ; Hút (1)
106   LD      M224  ; A D Plates C1
      ANI     M100  ; Manual
      OR      M115  ; MAN_ Hạ_Tấm_(1)
      OUT     Y032  ; Hạ_Tấm_(1)
110   LD      M225  ; A U Plates C1
      ANI     M100  ; Manual
      OR      M116  ; MAN_Nâng_Tấm_(1)
      OUT     Y033  ; Nâng_Tấm_(1)
114   LD      M226  ; A U Cyl Rotate_C1
      ANI     M100  ; Manual
      OR      M117  ; MAN_Nâng_Cụm_Xoay_(1)
      OUT     Y034  ; Nâng_Cụm_Xoay_(1)
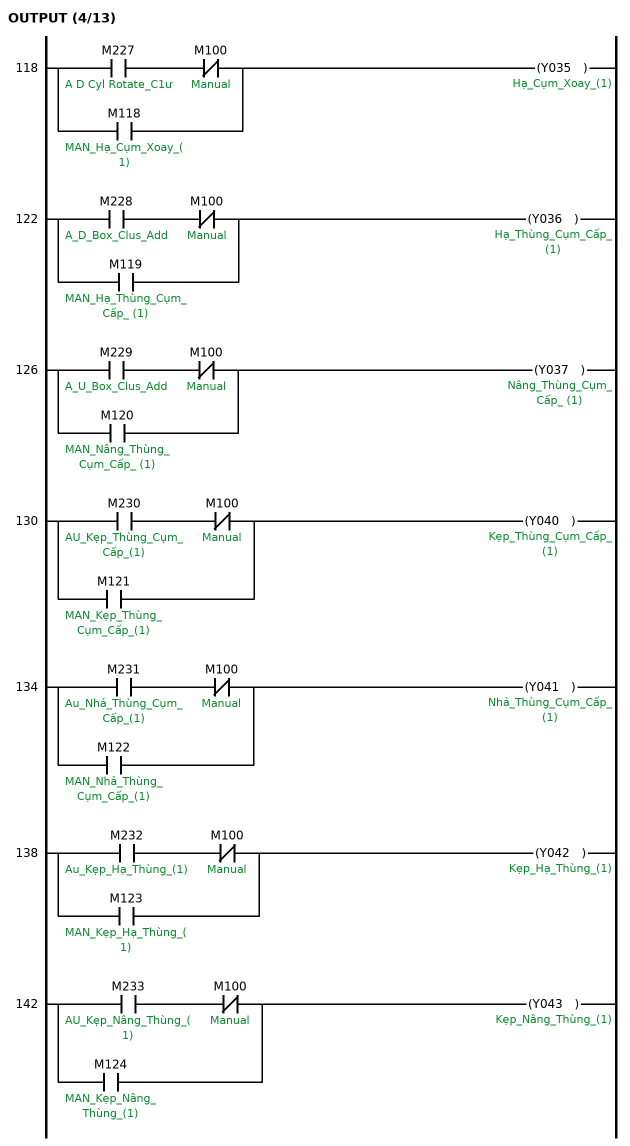
118   LD      M227  ; A D Cyl Rotate_C1ư
      ANI     M100  ; Manual
      OR      M118  ; MAN_Hạ_Cụm_Xoay_(1)
      OUT     Y035  ; Hạ_Cụm_Xoay_(1)
122   LD      M228  ; A_D_Box_Clus_Add
      ANI     M100  ; Manual
      OR      M119  ; MAN_Hạ_Thùng_Cụm_Cấp_ (1)
      OUT     Y036  ; Hạ_Thùng_Cụm_Cấp_ (1)
126   LD      M229  ; A_U_Box_Clus_Add
      ANI     M100  ; Manual
      OR      M120  ; MAN_Nâng_Thùng_Cụm_Cấp_ (1)
      OUT     Y037  ; Nâng_Thùng_Cụm_Cấp_ (1)
130   LD      M230  ; AU_Kẹp_Thùng_Cụm_Cấp_(1)
      ANI     M100  ; Manual
      OR      M121  ; MAN_Kẹp_Thùng_Cụm_Cấp_(1)
      OUT     Y040  ; Kẹp_Thùng_Cụm_Cấp_(1)
134   LD      M231  ; Au_Nhả_Thùng_Cụm_Cấp_(1)
      ANI     M100  ; Manual
      OR      M122  ; MAN_Nhả_Thùng_Cụm_Cấp_(1)
      OUT     Y041  ; Nhả_Thùng_Cụm_Cấp_(1)
138   LD      M232  ; Au_Kẹp_Hạ_Thùng_(1)
      ANI     M100  ; Manual
      OR      M123  ; MAN_Kẹp_Hạ_Thùng_(1)
      OUT     Y042  ; Kẹp_Hạ_Thùng_(1)
142   LD      M233  ; AU_Kẹp_Nâng_Thùng_(1)
      ANI     M100  ; Manual
      OR      M124  ; MAN_Kẹp_Nâng_Thùng_(1)
      OUT     Y043  ; Kẹp_Nâng_Thùng_(1)
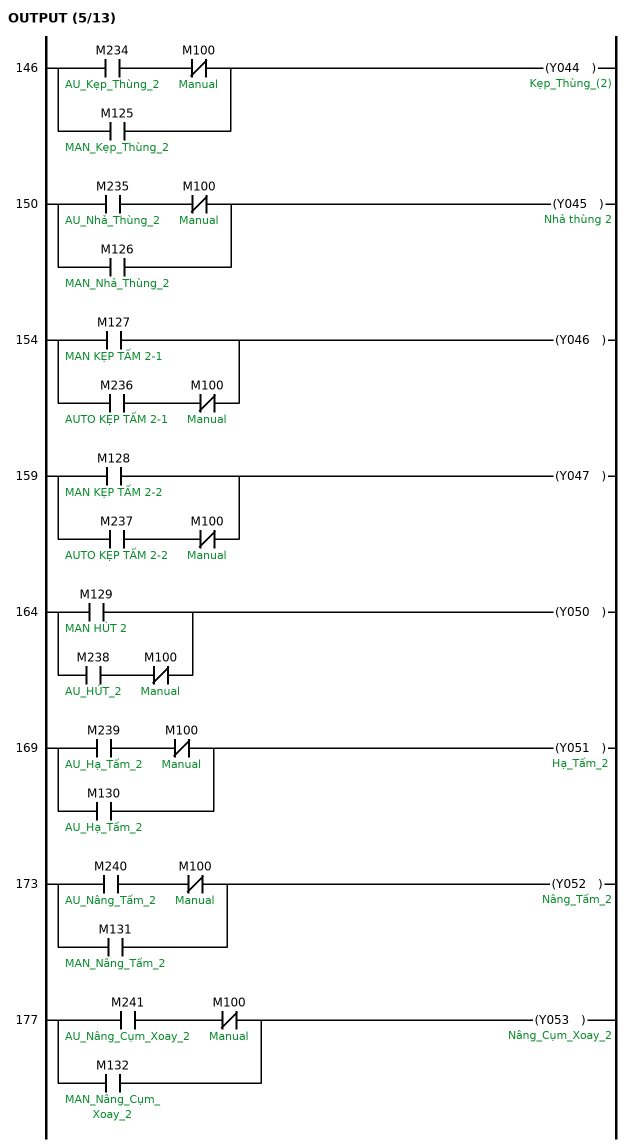
146   LD      M234  ; AU_Kẹp_Thùng_2
      ANI     M100  ; Manual
      OR      M125  ; MAN_Kẹp_Thùng_2
      OUT     Y044  ; Kẹp_Thùng_(2)
150   LD      M235  ; AU_Nhả_Thùng_2
      ANI     M100  ; Manual
      OR      M126  ; MAN_Nhả_Thùng_2
      OUT     Y045  ; Nhả thùng 2
154   LD      M127  ; MAN KẸP TẤM 2-1
      LD      M236  ; AUTO KẸP TẤM 2-1
      ANI     M100  ; Manual
      ORB
      OUT     Y046
159   LD      M128  ; MAN KẸP TẤM 2-2
      LD      M237  ; AUTO KẸP TẤM 2-2
      ANI     M100  ; Manual
      ORB
      OUT     Y047
164   LD      M129  ; MAN HÚT 2
      LD      M238  ; AU_HÚT_2
      ANI     M100  ; Manual
      ORB
      OUT     Y050
169   LD      M239  ; AU_Hạ_Tấm_2
      ANI     M100  ; Manual
      OR      M130  ; AU_Hạ_Tấm_2
      OUT     Y051  ; Hạ_Tấm_2
173   LD      M240  ; AU_Nâng_Tấm_2
      ANI     M100  ; Manual
      OR      M131  ; MAN_Nâng_Tấm_2
      OUT     Y052  ; Nâng_Tấm_2
177   LD      M241  ; AU_Nâng_Cụm_Xoay_2
      ANI     M100  ; Manual
      OR      M132  ; MAN_Nâng_Cụm_Xoay_2
      OUT     Y053  ; Nâng_Cụm_Xoay_2
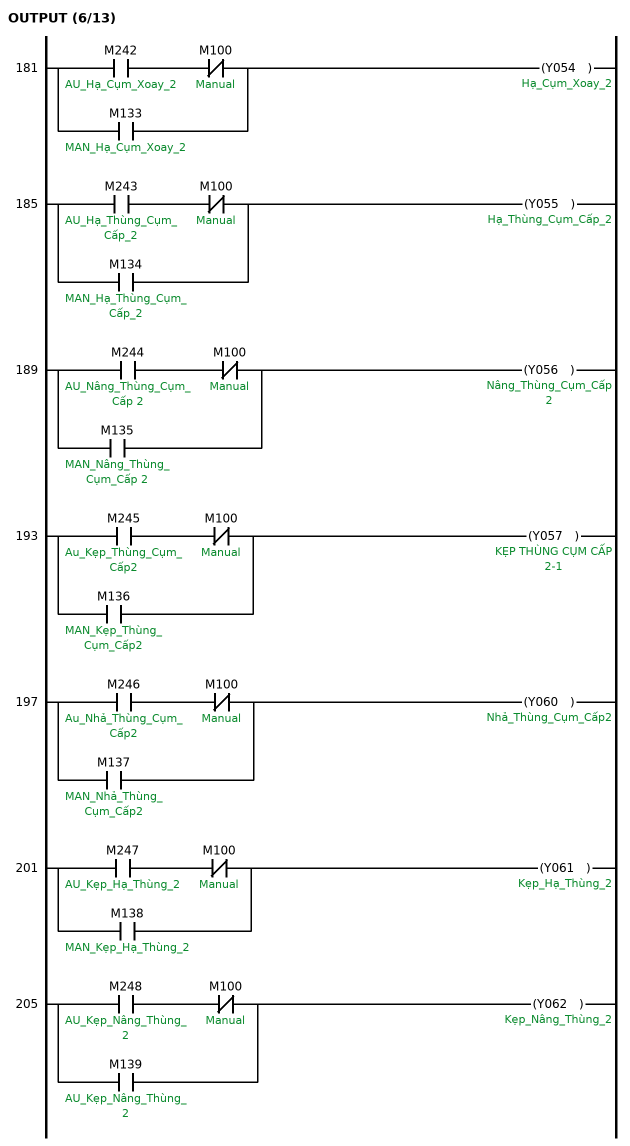
181   LD      M242  ; AU_Hạ_Cụm_Xoay_2
      ANI     M100  ; Manual
      OR      M133  ; MAN_Hạ_Cụm_Xoay_2
      OUT     Y054  ; Hạ_Cụm_Xoay_2
185   LD      M243  ; AU_Hạ_Thùng_Cụm_Cấp_2
      ANI     M100  ; Manual
      OR      M134  ; MAN_Hạ_Thùng_Cụm_Cấp_2
      OUT     Y055  ; Hạ_Thùng_Cụm_Cấp_2
189   LD      M244  ; AU_Nâng_Thùng_Cụm_Cấp 2
      ANI     M100  ; Manual
      OR      M135  ; MAN_Nâng_Thùng_Cụm_Cấp 2
      OUT     Y056  ; Nâng_Thùng_Cụm_Cấp 2
193   LD      M245  ; Au_Kẹp_Thùng_Cụm_Cấp2
      ANI     M100  ; Manual
      OR      M136  ; MAN_Kẹp_Thùng_Cụm_Cấp2
      OUT     Y057  ; KẸP THÙNG CỤM CẤP 2-1
197   LD      M246  ; Au_Nhả_Thùng_Cụm_Cấp2
      ANI     M100  ; Manual
      OR      M137  ; MAN_Nhả_Thùng_Cụm_Cấp2
      OUT     Y060  ; Nhả_Thùng_Cụm_Cấp2
201   LD      M247  ; AU_Kẹp_Hạ_Thùng_2
      ANI     M100  ; Manual
      OR      M138  ; MAN_Kẹp_Hạ_Thùng_2
      OUT     Y061  ; Kẹp_Hạ_Thùng_2
205   LD      M248  ; AU_Kẹp_Nâng_Thùng_2
      ANI     M100  ; Manual
      OR      M139  ; AU_Kẹp_Nâng_Thùng_2
      OUT     Y062  ; Kẹp_Nâng_Thùng_2
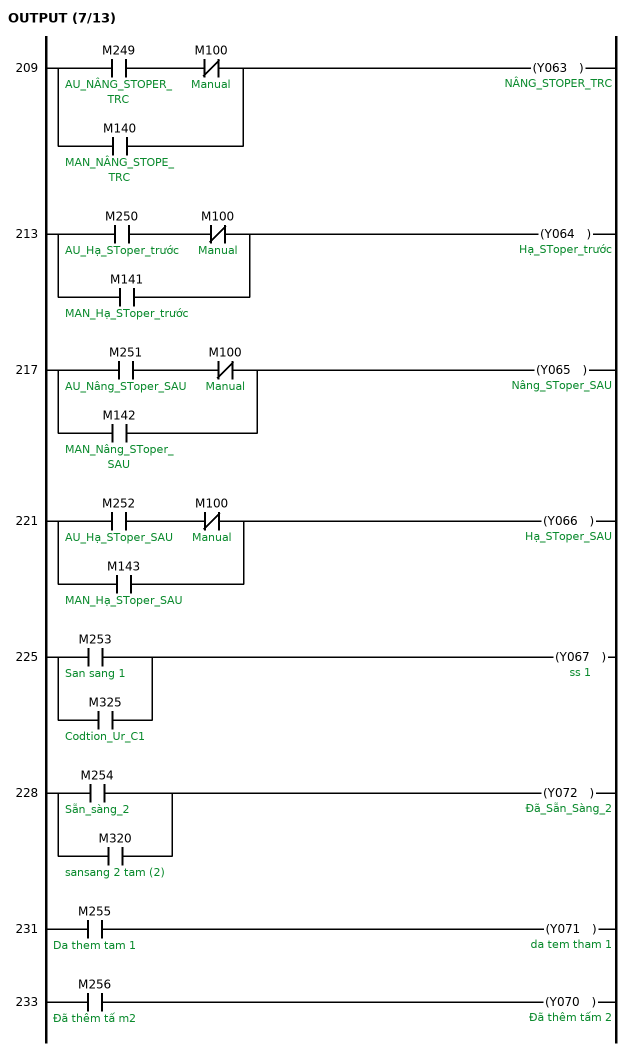
209   LD      M249  ; AU_NÂNG_STOPER_TRC
      ANI     M100  ; Manual
      OR      M140  ; MAN_NÂNG_STOPE_TRC
      OUT     Y063  ; NÂNG_STOPER_TRC
213   LD      M250  ; AU_Hạ_SToper_trước
      ANI     M100  ; Manual
      OR      M141  ; MAN_Hạ_SToper_trước
      OUT     Y064  ; Hạ_SToper_trước
217   LD      M251  ; AU_Nâng_SToper_SAU
      ANI     M100  ; Manual
      OR      M142  ; MAN_Nâng_SToper_SAU
      OUT     Y065  ; Nâng_SToper_SAU
221   LD      M252  ; AU_Hạ_SToper_SAU
      ANI     M100  ; Manual
      OR      M143  ; MAN_Hạ_SToper_SAU
      OUT     Y066  ; Hạ_SToper_SAU
225   LD      M253  ; San sang 1
      OR      M325  ; Codtion_Ur_C1
      OUT     Y067  ; ss 1
228   LD      M254  ; Sẵn_sàng_2
      OR      M320  ; sansang 2 tam (2)
      OUT     Y072  ; Đã_Sẵn_Sàng_2
231   LD      M255  ; Da them tam 1
      OUT     Y071  ; da tem tham 1
233   LD      M256  ; Đã thêm tấ m2
      OUT     Y070  ; Đã thêm tấm 2
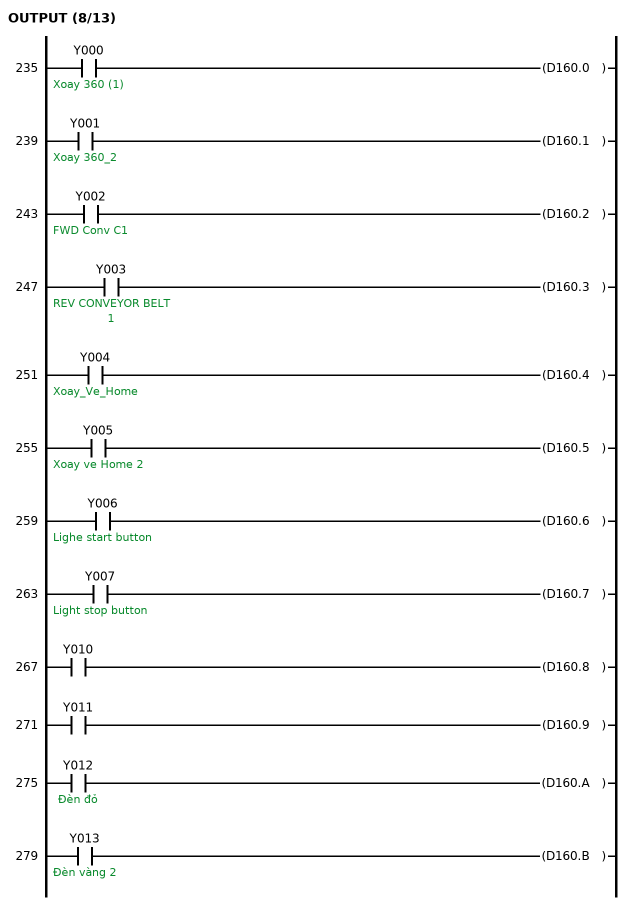
235   LD      Y000  ; Xoay 360 (1)
      OUT     D160.0
239   LD      Y001  ; Xoay 360_2
      OUT     D160.1
243   LD      Y002  ; FWD Conv C1
      OUT     D160.2
247   LD      Y003  ; REV CONVEYOR BELT 1
      OUT     D160.3
251   LD      Y004  ; Xoay_Ve_Home
      OUT     D160.4
255   LD      Y005  ; Xoay ve Home 2
      OUT     D160.5
259   LD      Y006  ; Lighe start button
      OUT     D160.6
263   LD      Y007  ; Light stop button
      OUT     D160.7
267   LD      Y010
      OUT     D160.8
271   LD      Y011
      OUT     D160.9
275   LD      Y012  ; Đèn đỏ
      OUT     D160.A
279   LD      Y013  ; Đèn vàng 2
      OUT     D160.B
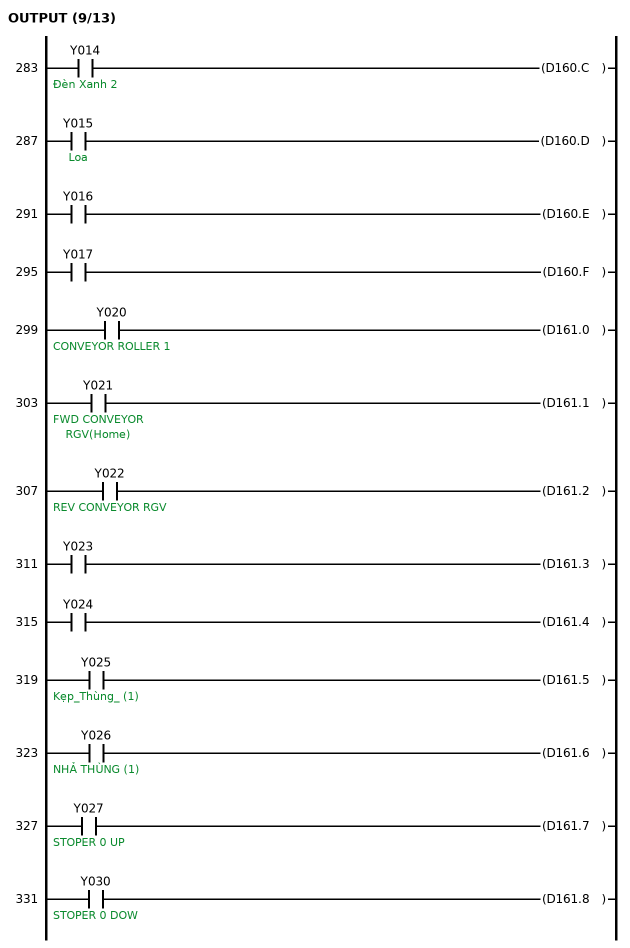
283   LD      Y014  ; Đèn Xanh 2
      OUT     D160.C
287   LD      Y015  ; Loa
      OUT     D160.D
291   LD      Y016
      OUT     D160.E
295   LD      Y017
      OUT     D160.F
299   LD      Y020  ; CONVEYOR ROLLER 1
      OUT     D161.0
303   LD      Y021  ; FWD CONVEYOR RGV(Home)
      OUT     D161.1
307   LD      Y022  ; REV CONVEYOR RGV
      OUT     D161.2
311   LD      Y023
      OUT     D161.3
315   LD      Y024
      OUT     D161.4
319   LD      Y025  ; Kẹp_Thùng_ (1)
      OUT     D161.5
323   LD      Y026  ; NHẢ THÙNG (1)
      OUT     D161.6
327   LD      Y027  ; STOPER 0 UP
      OUT     D161.7
331   LD      Y030  ; STOPER 0 DOW
      OUT     D161.8
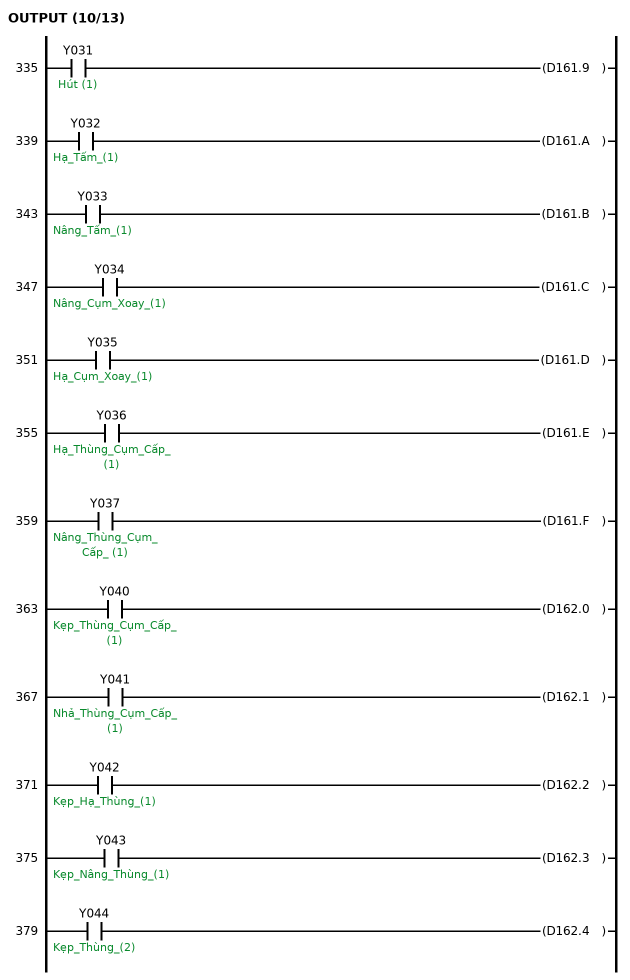
335   LD      Y031  ; Hút (1)
      OUT     D161.9
339   LD      Y032  ; Hạ_Tấm_(1)
      OUT     D161.A
343   LD      Y033  ; Nâng_Tấm_(1)
      OUT     D161.B
347   LD      Y034  ; Nâng_Cụm_Xoay_(1)
      OUT     D161.C
351   LD      Y035  ; Hạ_Cụm_Xoay_(1)
      OUT     D161.D
355   LD      Y036  ; Hạ_Thùng_Cụm_Cấp_ (1)
      OUT     D161.E
359   LD      Y037  ; Nâng_Thùng_Cụm_Cấp_ (1)
      OUT     D161.F
363   LD      Y040  ; Kẹp_Thùng_Cụm_Cấp_(1)
      OUT     D162.0
367   LD      Y041  ; Nhả_Thùng_Cụm_Cấp_(1)
      OUT     D162.1
371   LD      Y042  ; Kẹp_Hạ_Thùng_(1)
      OUT     D162.2
375   LD      Y043  ; Kẹp_Nâng_Thùng_(1)
      OUT     D162.3
379   LD      Y044  ; Kẹp_Thùng_(2)
      OUT     D162.4
